TYPE ST_HEATER_SETTINGS :
STRUCT
	targetTemperature:		REAL;
END_STRUCT
END_TYPE

(* stored: Version 1.1.0.1
   DUT ST_HEATER_SETTINGS: Id {d9ba9ecf-ff30-4fb2-9564-5ba2698082b8} *)
